(*======================================================================================================================================*)
(*fb_RS485ComCheck:	Einfacher Universal Ping Baustein um von allerlei Geräten von haus-bus.de Kommunikation zu Checken über RS485 
	In Diesem Fall ist es für einen Taster (BTN) bei einem Relais sollte es (OUT) sein*)
(*
Date          	| Version    	| created under        	| Author          	| Remark *)
(*====================================================================================================================================================*)
(*05/05/2025   	| 1.00      		| TC3		  		| N.Kersting       | first release *)
(*06/05/2025   	| 1.01      		| TC3		  		| N.Kersting       | Bugfix Timeouts werden besser ausgewertet *)
(*07/05/2025   	| 1.02      		| TC3		  		| N.Kersting       | Bug in Schritt 2 behoben (weiter, wenn nicht Busy) *)
(*09/05/2025   	| 1.03      		| TC3		  		| N.Kersting       | Counter für verbindungsversuche inkl. erneut senden *)
(*10/05/2025   	| 1.04      		| TC3		  		| N.Kersting       | Umrüstung Auf Externen Fifo  *)
(*12/05/2025   	| 1.05      		| TC3		  		| N.Kersting       | Verriegelung über I_bStart, damit nich gesendet werden kann wenn nicht Freigegeben  *)
(*14/05/2025   	| 1.06      		| TC3		  		| N.Kersting       | Ausgänge ergänzt für Done  *)
(*====================================================================================================================================================*)
FUNCTION_BLOCK fb_RS485ComCheck_1
VAR_INPUT
	I_FifoID			:INT;
	I_bExecute			:BOOL;							(* Aktiviert den Baustein *)
	I_bStart			:BOOL;							(* Startet das Senden des Pings *)
	I_tPingIntervall	:TIME := T#5S;					(* Intervall Zeit wann die Kommunikation geprüft werden soll *)
	I_tPingTimeout		:TIME := T#2S;					(* Zeit, bis der Ping zurück gekommen sein muss *)
	I_diID				:DINT;							(* Device ID *)
	I_sPingSymbol		:STRING :='.BTN.';				(* Symbol, welches als Ping genutzt werden soll *)
	I_iInstID			:INT := 17;						(* Instanz ID *)
	I_sStartZeichen		:BYTE := 16#FD;					(* Startzeichen Präfix *)
	I_sEndZeichen		:BYTE := 16#FE;					(* Endzeichen Suffix *)
	I_StringReceived	:STRING(255);					(* Empfangener String *)
	I_iMaxPingTry		:INT := 5;
	I_bTasterMode		:BOOL;							(* Wenn ein Taster Abgefragt wird, gibt es die Besonderheit, dass dieser Selbst Signale Sendet (Helligkeit, temperatur usw. *)
END_VAR
VAR_OUTPUT
	Q_sSend				:STRING(255);
	Q_bBusy 			:BOOL;
	Q_bSendDone			:BOOL;
	Q_sState			:STRING;
	Q_bComOk			:BOOL;
	Q_bTimeout			:BOOL;
	Q_bError			:BOOL;
END_VAR
VAR
	sStringSend			:STRING;
	fbBusPingEvent		:ARRAY[1..6] OF fb_BusPingEvent;
	
	tonIntervall		:ton;
	tonTimeout			:ton;
	tonRecevieAutoReset	:ton;
	
	iStepReceive		:INT;
	iStep				:INT;
	icntComTry			:INT;
	iMaxComTry			:INT := 5;
	i					:INT;
	icntSymbole			:INT;
	
	bSend				:BOOL;
	bReceived			:BOOL;
	bCOMMem				:BOOL;
END_VAR

iMaxComTry :=	I_iMaxPingTry;

(* Intervall timer *)
tonIntervall(
	PT := I_tPingIntervall);
	
(* Timeout timer *)
tonTimeout(
	PT := I_tPingTimeout);
	
(* Ping String ertsllen *)
sStringSend:=	CONCAT(F_ToCHR(I_sStartZeichen),DINT_TO_STRING(I_diID));
sStringSend:=	CONCAT(sStringSend,I_sPingSymbol);
sStringSend:=	CONCAT(sStringSend,INT_TO_STRING(I_iInstID));
sStringSend:=	CONCAT(sStringSend,'.gSTATUS');
sStringSend:=	CONCAT(sStringSend,F_ToCHR(I_sEndZeichen));

IF NOT I_bExecute 
	AND NOT I_bTasterMode
THEN
	Q_bComOk := FALSE;
	Q_bTimeout := FALSE;
	tonIntervall.IN := FALSE;
	tonTimeout.IN := FALSE;
	sStringSend:= '';
	bSend := FALSE;
	iStep := 0;
ELSE
	ac01_Send();
END_IF

ACTION ac01_Send:
(* Sende Schrittkette *)
			
CASE iStep OF
(*=========================================================*)	
0:	Q_sState := ' INIT';
	tonIntervall.IN := FALSE;
	tonTimeout.IN := FALSE;
	bCOMMem := FALSE;
	bSend := FALSE;
	Q_bBusy := FALSE;
	Q_sSend := '';
	
	IF I_bExecute
		AND I_bStart
	THEN
		Q_bSendDone := FALSE;
		Q_bBusy := TRUE;
		iStep := iStep +1;
	ELSIF
		NOT I_bExecute
		AND I_bTasterMode
	THEN
		iStep := 10;
	END_IF

(*=========================================================*)	
1:	Q_sState := 'Starte Sendebefehl';
	
	IF GVL_RS485FiFoSend.bSendDoneFiFo[I_FifoID]
	THEN
		tonTimeout.IN := TRUE;
		Q_sSend := sStringSend;
	END_IF
	IF NOT GVL_RS485FiFoSend.bSendDoneFiFo[I_FifoID]
	THEN
		tonTimeout.IN := FALSE;
		iStep := iStep +1;
	ELSIF
		tonTimeout.Q
	THEN
		tonTimeout.IN := FALSE;
		Q_sState := 'Timeout Send Busy';
		iStep := -1;
	END_IF
	
(*=========================================================*)	
2:	Q_sState := 'Auswertung Senden';
	bSend := FALSE;	
	tonTimeout.IN := TRUE;
	
	IF GVL_RS485FiFoSend.bSendDoneFiFo[I_FifoID]
	THEN
		Q_sSend := '';
		Q_bSendDone := TRUE;
		tonTimeout.IN := FALSE;
		iStep := iStep +1;
	ELSIF
		tonTimeout.Q
	THEN
		Q_sState := 'Timeout Send Done';
		iStep := -2;
	END_IF
		
(*=========================================================*)	
3:	Q_sState := 'Warte auf Empfang';
	tonTimeout.IN := TRUE;
	
	IF tonTimeout.Q
	THEN
		(* Kommunikations versuche *)
		IF icntComTry <iMaxComTry
		THEN
			icntComTry := icntComTry +1;
			iStep := 5;				(* Erneut Senden *)
		ELSE
			Q_sState := 'Timeout kein Ping Empfangen';
			Q_bComOk := FALSE;
			Q_bTimeout := TRUE;
			iStep := -4;	(* Erneut Empfangen *)
		END_IF
	ELSE
		
		IF	bCOMMem
		THEN
			bCOMMem := FALSE;
			iStep := iStep+1;		(* Telegram erhalten *)
		END_IF
	END_IF
	
(*=========================================================*)	
4:	Q_sState := 'Ping Empfangen, Warte auf Intervall';
	tonIntervall.IN := TRUE;
	Q_bComOk := TRUE;
	Q_bTimeout := FALSE;
	
	IF tonIntervall.Q
		AND I_bStart
	THEN
		icntComTry := 0;	(* Wenn die Verbindung wieder da ist dürfen die Versuche gelöscht werden *)
		iStep := 0;
	END_IF

(*=========================================================*)	
5:	Q_sState := 'Ping nicht Empfangen, Warte auf Intervall';
	tonIntervall.IN := TRUE;
	
	IF tonIntervall.Q
		AND I_bStart
	THEN
		iStep := 0;
	END_IF

(*=========================================================*)	
10:	Q_sState := 'Warten Auf Automatischen Ping vom Taster';
	tonIntervall.IN := TRUE;
	
	IF tonIntervall.Q
		AND I_bStart
	THEN
		Q_bComOk := FALSE;
		iStep := 0;
	ELSE
		IF bCOMMem
		THEN
			tonIntervall.IN := FALSE;
			Q_bComOk := TRUE;
			iStep := 0;
		END_IF
	END_IF	
ELSE
	tonIntervall.IN := TRUE;
	tonTimeout.IN := FALSE;
	Q_bComOk := FALSE;
	bSend := FALSE;
	Q_bBusy := FALSE;
	icntComTry := 0;
	Q_sSend := '';
	
	IF tonIntervall.Q
		AND I_bStart
	THEN
		iStep := 0;
	END_IF
END_CASE

IF I_bTasterMode
THEN
	icntSymbole := 0;
	(* Durchgehend Checken ob Ping kommt *)
	FOR i := 1 TO 6 BY 1 DO 
		fbBusPingEvent[i](
			I_bReset := 			FALSE,
			I_sID:= 				DINT_TO_STRING(I_diID ), 
			I_iInstID:=				I_iInstID -1 +i,	
			I_sReceivedString:= 	I_StringReceived, 
			I_bTasterMode := 		TRUE,
			Q_bOut=> 				);
			
		IF fbBusPingEvent[i].Q_bOut
		THEN
			icntSymbole := icntSymbole +1;
		END_IF
	END_FOR
	
	IF iStep > 0
		AND icntSymbole >0
	THEN
		bCOMMem := TRUE;
	END_IF
ELSE
	(* Nur nach der einen ID Gucken *)
	fbBusPingEvent[1](
		I_bReset := 			FALSE,
		I_sID:= 				DINT_TO_STRING(I_diID ), 
		I_iInstID:=				I_iInstID,	
		I_sReceivedString:= 	I_StringReceived, 
		I_bTasterMode := 		FALSE,
		Q_bOut=> 				);
		
	IF iStep > 0
		AND fbBusPingEvent[1].Q_bOut
	THEN
		bCOMMem := TRUE;
	END_IF
END_IF
END_ACTION

END_FUNCTION_BLOCK

(* stored: Version 1.1.0.1, ProductVersion 3.1.4024.12
   POU fb_RS485ComCheck_1: Id {76148ca7-cd8f-458e-8701-480688e882bc}, SpecialFunc None
   Action ac01_Send: Id {239e4ad7-dc6a-460b-afb5-48a7f527635b} *)
